PROGRAM registradorLog
VAR
	i: INT;
	j: INT;
	k: INT;
END_VAR


IF gvl.logRegister19 <> '' THEN
	FOR i:=100 TO 1 BY -1 DO
		IF gvl_p.arrLogEstufa19[i] <> '' THEN
			gvl_p.arrLogEstufa19[i+1]:= gvl_p.arrLogEstufa19[i];
			gvl_p.arrLogEstufa19[i]:= '';
		END_IF
	END_FOR
	gvl_p.arrLogEstufa19[1]:= concat(gvl_p.arrLogEstufa19[1],gvl.sSystemDateTime);
	gvl_p.arrLogEstufa19[1]:= concat(gvl_p.arrLogEstufa19[1],'    ');
	gvl_p.arrLogEstufa19[1]:= concat(gvl_p.arrLogEstufa19[1],gvl.logRegister19);
	gvl.sCmdInsertLog:= 'INSERT INTO [dbo].[LogGeneral] ([HistoricalTime],[Description])VALUES($'$',$'$')';
	gvl.sCmdInsertLog:= insert(gvl.sCmdInsertLog,gvl.logRegister19,74);	
	gvl.sCmdInsertLog:= insert(gvl.sCmdInsertLog,gvl.sSystemDateTime,71);
	gvl.bInsertLog:=true;
	gvl.logRegister19:= '';
	
	
END_IF

END_PROGRAM

(* stored: Version 1.1.0.1, ProductVersion 3.1.4024.12
   POU registradorLog: Id {a508c4aa-10ae-4ca7-86e7-a9f98e066205}, SpecialFunc None *)
